INTERFACE I_PositioningHomingBuilder EXTENDS __System.IQueryInterface

METHOD BuildDefaultHomingCommand : HomingCommand
END_METHOD

METHOD BuildDirectHomingCommand : HomingCommand
END_METHOD

METHOD Cam : I_DefaultHomingBuilder
VAR_INPUT
	value : REFERENCE TO BOOL;
END_VAR
END_METHOD

METHOD ClearLag : I_PositioningHomingBuilder
END_METHOD

METHOD KeepLag : I_PositioningHomingBuilder
END_METHOD

METHOD Position : I_PositioningHomingBuilder
VAR_INPUT
	value : LREAL;
END_VAR
END_METHOD

METHOD ReferenceMode : I_DefaultHomingBuilder
VAR_INPUT
	value : EncoderReferenceMode;
END_VAR
END_METHOD

METHOD SearchDirection : I_DefaultHomingBuilder
VAR_INPUT
	value : Direction;
END_VAR
END_METHOD

METHOD SearchVelocity : I_DefaultHomingBuilder
VAR_INPUT
	value : LREAL;
END_VAR
END_METHOD

METHOD SyncDirection : I_DefaultHomingBuilder
VAR_INPUT
	value : Direction;
END_VAR
END_METHOD

METHOD SyncVelocity : I_DefaultHomingBuilder
VAR_INPUT
	value : LREAL;
END_VAR
END_METHOD

END_INTERFACE

(* stored: Version 1.1.0.1, ProductVersion 3.1.4026.13
   Itf I_PositioningHomingBuilder: Id {415b10b5-af07-0f72-3584-1972e285a25b}
   Method BuildDefaultHomingCommand: Id {0244a079-57b6-032a-2be7-5b7be1987cf5}
   Method BuildDirectHomingCommand: Id {8544b382-d7b7-0a47-2667-0721e7869f3d}
   Method Cam: Id {c942ca77-cc81-08b3-3ce6-ecfa33601a2e}
   Method ClearLag: Id {b8e3e26a-ec28-018b-22ed-6d821d837a12}
   Method KeepLag: Id {20ffe9af-ac17-0a55-144c-ed95ca7bb53f}
   Method Position: Id {3dd70a34-1c87-0933-3cbe-b8d3b2f1587d}
   Method ReferenceMode: Id {1e534404-5d70-01e3-2097-e484650b1ed9}
   Method SearchDirection: Id {3cbab8b1-b379-0388-072f-eafbe47da304}
   Method SearchVelocity: Id {f38c3e5f-8d3c-0f61-13de-0f82a85a7522}
   Method SyncDirection: Id {adc4aba0-c1e6-0812-3de0-82d15bee5f19}
   Method SyncVelocity: Id {1e3cde5a-a5f9-01a4-3610-1515305acad5} *)
